PROGRAM Alarm_Display_ST
VAR
END_VAR

END_PROGRAM

(* stored: Version 1.1.0.1, ProductVersion 3.1.4024.0
   POU Alarm_Display_ST: Id {4dff6505-02b3-42cb-a57d-8b2cccbd18bf}, SpecialFunc None *)
